Staubli VAL3: robot2PC.pgx

program robot2PC()
begin
  //清空缓存
  clearBuffer(sktoPC)
  //设置终止符 $
  sioCtrl(sktoPC,"endOfString",36)
  do
    sktoPC="run"
    sDataPC=sktoPC
    _bVisionOK=true
    delay(1)
  until false
end
